TYPE E_MotionTrajectory :
(
	Ramp := 0,
	Sine := 1,
	fUTest := 2
);
END_TYPE

(* stored: Version 1.1.0.1
   DUT E_MotionTrajectory: Id {a50a2702-f044-4930-85d0-69fbdaa9544e} *)
